FUNCTION_BLOCK FB_TemperatureSensor
VAR_INPUT
END_VAR
VAR_OUTPUT
END_VAR
VAR
END_VAR

END_FUNCTION_BLOCK

(* stored: Version 1.1.0.1, ProductVersion 3.1.4024.9
   POU FB_TemperatureSensor: Id {aa82beeb-f8d4-4ab1-8220-d0c7217097c1}, SpecialFunc None *)
